Yaskawa INFORM job: TEST-BELOW.JBI

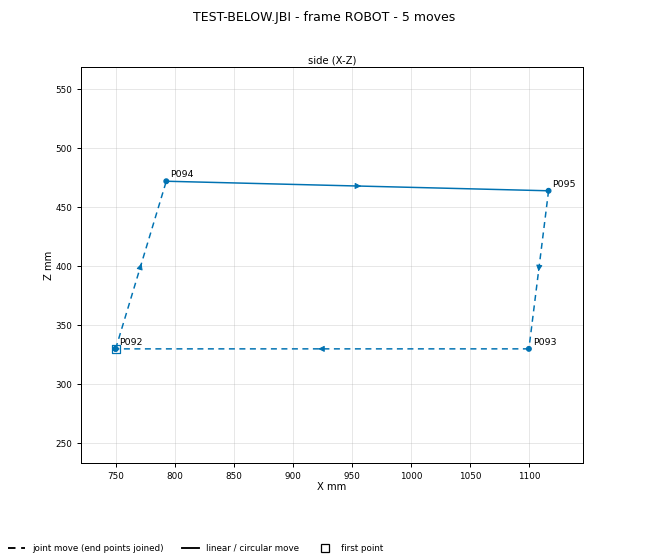
[picture p0: tool path of TEST-BELOW.JBI in frame ROBOT, 5 of 5 moves have a stored position in this frame; points joined in program order, loops and branches not executed]
/JOB
//NAME TEST-BELOW
///FOLDERNAME FOLDER001
//POS
///NPOS 2,0,0,4,0,0
///USER 15
///TOOL 1
///POSTYPE USER
///RECTAN
///RCONF 0,0,0,0,1,0,0,0,0,0,0,0,0,0,0,0,0,0,0,0,0,0,0,0
C00000=5.957,15.445,-75.515,0.0000,10.0000,0.0000
///RCONF 0,0,0,0,0,0,0,0,0,0,0,0,0,0,0,0,0,0,0,0,0,0,0,0
C00001=6.407,-26.777,-97.787,-0.0035,10.0001,0.0367
///POSTYPE ROBOT
P00092=750.003,161.812,330.004,0.1640,10.0066,0.1393
P00093=1100.002,161.807,330.008,0.1639,24.9999,0.1388
P00094=792.896,160.291,471.972,0.0813,10.0064,0.0684
P00095=1116.664,160.280,463.887,0.0787,10.0067,0.0664
//INST
///DATE 2025/10/03 10:09
///ATTR SC,RW,RJ
////FRAME USER 15
///GROUP1 RB1
///LVARS 20,20,20,0,0,0,0,0
NOP
'ROOT
SFTOF
MACRO1 MJ#(2) ARGF2.4 ARGF1.0 ARGF16.0
MACRO1 MJ#(1) ARGF0.0 ARGF0.0 ARGF0.0 ARGF0.0 ARGF0.0 ARGF0.0
REFP 1 C00000
REFP 2 C00001
MOVJ P092 VJ=15.00 PL=3
MOVJ P094 VJ=15.00 PL=0
WVON AMP=D080 FREQ=D081 ANGL=D082
WVADJ STD=4.000 ST=4.000 END=4.000 LEN=400.000 ADJMD=0
MOVL P095 V=58.3 PL=0
WVOF
MOVJ P093 VJ=15.00 PL=3
MOVJ P092 VJ=15.00 PL=3
END
